FUNCTION_BLOCK Test_AssertEquals_WORD EXTENDS TUnitTestBase
VAR
    AssertionUnderTest : TAssertion(AssertionListenerMock);
    AssertionListenerMock : TAssertionListenerMock;
    WORD_Variable : WORD;
END_VAR

AssertionListenerMock.AssertionFailed  := FALSE;
AssertionListenerMock.AssertionMessage := '';
AssertionListenerMock.ExpectedAsString := '';
AssertionListenerMock.ActualAsString   := '';

// Test the assertion...
WORD_Variable := 1111;

AssertionUnderTest.AssertEquals_WORD(
    Expected := 2222, // deliberately different to test the assertion
    Actual   := WORD_Variable,
    VariableName := 'WORD_Variable');
 
// Check the assertion worked...    
Assertion.AssertEquals_BOOL(
    Expected := TRUE,
    Actual   := AssertionListenerMock.AssertionFailed,
    VariableName := 'AssertionListenerMock.AssertionFailed');

// Check the assertion messages...    
Assertion.AssertEquals_STRING(
    Expected := 'AssertEquals_WORD failed in AssertionListenerMock: Value "WORD_Variable"',
    Actual   := AssertionListenerMock.AssertionMessage,
    VariableName := 'AssertionListenerMock.AssertionMessage');

Assertion.AssertEquals_STRING(
    Expected := '  Expected = 2222',
    Actual   := AssertionListenerMock.ExpectedAsString,
    VariableName := 'AssertionListenerMock.ExpectedAsString');

Assertion.AssertEquals_STRING(
    Expected := '  Actual   = 1111',
    Actual   := AssertionListenerMock.ActualAsString,
    VariableName := 'AssertionListenerMock.ActualAsString');


TestFinished();

END_FUNCTION_BLOCK

(* stored: Version 1.1.0.1, ProductVersion 3.1.4024.4
   POU Test_AssertEquals_WORD: Id {302df836-097e-4453-af80-790301b29cf5}, SpecialFunc None *)
